TYPE StringByteArray :

UNION
	bArray: ARRAY[0..254] OF BYTE;
	sString: STRING(255);
END_UNION

END_TYPE

(* stored: Version 1.1.0.1
   DUT StringByteArray: Id {74ac9c91-8dd0-4804-83eb-55aba09ae987} *)
